FUNCTION_BLOCK PID (* PID FB *)
  (* Standard: 61499-2 *)
  (* Version 1.0, 2026-04-19, Thomas Mayr *)
  PACKAGE eclipse4diac::controlengineering;
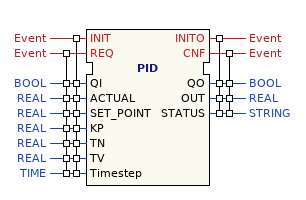
  EVENT_INPUT
    INIT WITH QI, ACTUAL, SET_POINT, KP, TN, TV, Timestep; (* Initialize controller *)
    REQ WITH QI, ACTUAL, SET_POINT, KP, TN, TV, Timestep; (* Execute control step *)
  END_EVENT
  EVENT_OUTPUT
    INITO WITH QO, OUT, STATUS; (* Initialization done *)
    CNF WITH QO, OUT, STATUS; (* Calculation done *)
  END_EVENT
  VAR_INPUT
    QI : BOOL; (* Enable input *)
    ACTUAL : REAL; (* Process value *)
    SET_POINT : REAL; (* Setpoint *)
    KP : REAL; (* Proportional gain *)
    TN : REAL; (* Integral time [s] *)
    TV : REAL; (* Derivative time [s] *)
    Timestep : TIME; (* Sampling time (cycle time) *)
  END_VAR
  VAR_OUTPUT
    QO : BOOL; (* Enable output *)
    OUT : REAL; (* Controller output (0..100%) *)
    STATUS : STRING; (* Service Status *)
  END_VAR
  VAR
    ERR : REAL;
    ERR_OLD : REAL;
    I_SUM : REAL;
    DT_SEC : REAL;
    D_TERM : REAL;
  END_VAR
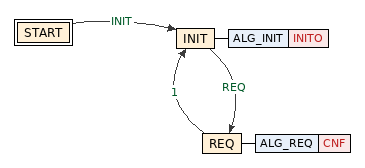
  EC_STATES
    START; (* Initial State *)
    INIT : ALG_INIT -> INITO;
    REQ : ALG_REQ -> CNF;
  END_STATES
  EC_TRANSITIONS
    START TO INIT := INIT;
    REQ TO INIT := 1;
    INIT TO REQ := REQ;
  END_TRANSITIONS
  ALGORITHM ALG_INIT IN ST:
QO := QI;
ERR := 0.0;
ERR_OLD := 0.0;
I_SUM := 0.0;
DT_SEC := 0.0;
D_TERM := 0.0;
OUT := 0.0;
  END_ALGORITHM
  ALGORITHM ALG_REQ IN ST:
QO := QI;

IF NOT QI THEN
	OUT := 0.0;
	I_SUM := 0.0;
	D_TERM := 0.0;
ELSE
	DT_SEC := LREAL_TO_REAL(TIME_IN_S_TO_LREAL(Timestep));
	IF DT_SEC <= 0.0 OR KP <= 0.0 THEN
		STATUS := 'Inputs out of Range';
		OUT := 0.0;
	ELSE
		STATUS := 'PID Active';
		ERR := SET_POINT - ACTUAL;

			(* I-Term *)
		IF TN > 0.0 THEN
			IF NOT ((OUT >= 100.0 AND ERR > 0.0) OR (OUT <= 0.0 AND ERR < 0.0)) THEN
				I_SUM := I_SUM + (KP * ERR * DT_SEC / TN);
			END_IF;
		ELSE
			I_SUM := 0.0;
		END_IF;

			(* D-Term *)
		IF TV > 0.0 THEN
			D_TERM := KP * TV * (ERR - ERR_OLD) / DT_SEC;
		ELSE
			D_TERM := 0.0;
		END_IF;

		OUT := KP * ERR + I_SUM + D_TERM;

		IF OUT > 100.0 THEN
			OUT := 100.0;
		ELSIF OUT < 0.0 THEN
			OUT := 0.0;
		END_IF;

		ERR_OLD := ERR;
	END_IF;
END_IF;
  END_ALGORITHM
END_FUNCTION_BLOCK
